(* PLC project poST.project, poSTIDE *)
(* stored: creationDateTime 2021-08-31T00:00:00.000000 *)

FUNCTION_BLOCK TON
  VAR_INPUT
    in : BOOL;
    pt : TIME;
  END_VAR
  VAR_OUTPUT
    q : BOOL;
    et : TIME;
  END_VAR

END_FUNCTION_BLOCK
